// TIA Portal project "aritmetik_islemler" (V18)

(* hardware
DEVICE "S7-1200 station_1"  S7-1200 Station
   slot 0: "Rack_0"  S7-1200 Rack  Rack  V1.0
   slot 1: "PLC_1"  CPU 1214C AC/DC/Rly  6ES7 214-1BG40-0XB0  V4.6
*)

// ===== PLC "PLC_1"  CPU 1214C AC/DC/Rly =====

VAR_GLOBAL   // PLC tag table "Default tag table"
   "Tag_1" AT %I0.0 : Bool;
   "Tag_2" AT %Q0.0 : Bool;
   "Tag_3" AT %MD0 : DWord;
   "Tag_4" AT %MD8 : Real;
   "Tag_5" AT %MW2 : Int;
   "Tag_6" AT %I0.1 : Bool;
   "Tag_7" AT %M4.0 : Bool;
   "Tag_8" AT %MW8 : Int;
   "Tag_9" AT %MD16 : Real;
   "Tag_10" AT %MD12 : Real;
   "Tag_11" AT %MD24 : Real;
   "Tag_12" AT %MD20 : Real;
   "Tag_13" AT %MD10 : DWord;
END_VAR

DATA_BLOCK "Data_block_1"   // DB1
{ S7_Optimized_Access := 'TRUE' }
VERSION : 0.1
   VAR
      "A" : LReal;
      "B" : LReal;
   END_VAR
BEGIN
END_DATA_BLOCK

ORGANIZATION_BLOCK "Main"   // OB1, LAD, ProgramCycle
TITLE = "Main Program Sweep (Cycle)"
{ S7_Optimized_Access := 'TRUE' }
VERSION : 0.1
   VAR_INPUT
      Initial_Call : Bool;   // Initial call of this OB
      Remanence : Bool;   // =True, if remanent data are available
   END_VAR
   VAR_TEMP   // added for the SCL form of the ladder/FBD networks
      _w1 : Bool;
   END_VAR
BEGIN

REGION Network 1
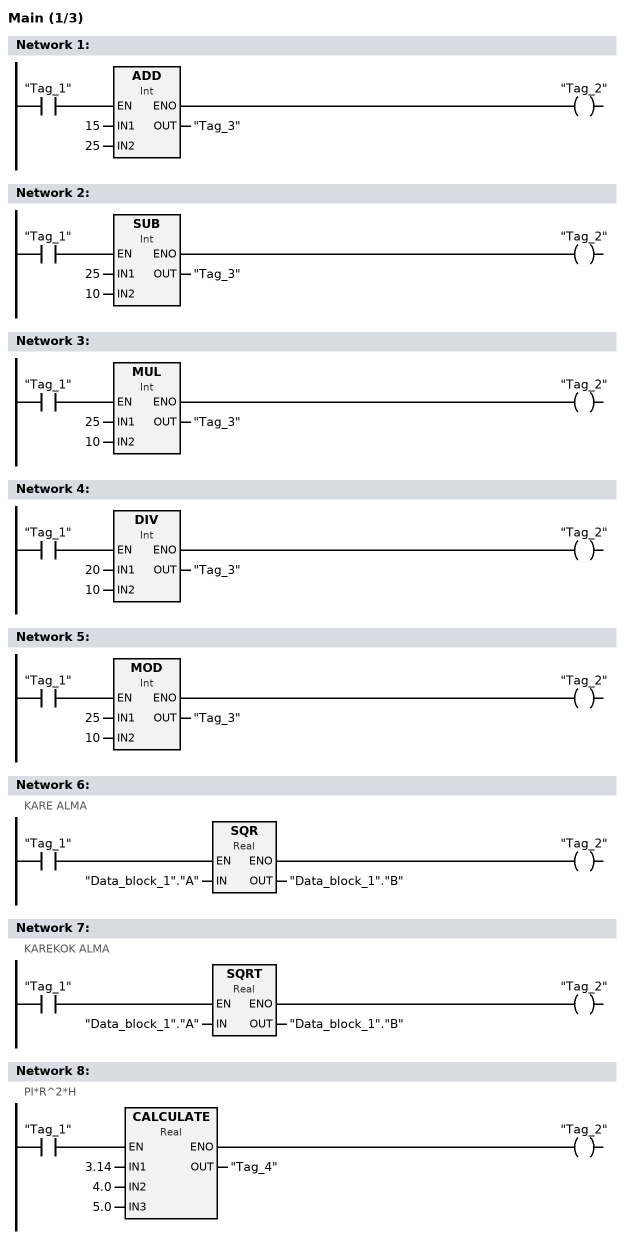
   RUNG wire#powerrail
      Contact( "Tag_1" )
      { S7_Templates := "SrcType := Int" } Add(in1 := 15, in2 := 25, out => "Tag_3")
      Coil( "Tag_2" )
   END_RUNG
   // the same network as SCL:
   IF "Tag_1" THEN "Tag_3" := 15 + 25; END_IF;
   "Tag_2" := "Tag_1";
END_REGION

REGION Network 2
   RUNG wire#powerrail
      Contact( "Tag_1" )
      { S7_Templates := "SrcType := Int" } Sub(in1 := 25, in2 := 10, out => "Tag_3")
      Coil( "Tag_2" )
   END_RUNG
   // the same network as SCL:
   IF "Tag_1" THEN "Tag_3" := 25 - 10; END_IF;
   "Tag_2" := "Tag_1";
END_REGION

REGION Network 3
   RUNG wire#powerrail
      Contact( "Tag_1" )
      { S7_Templates := "SrcType := Int" } Mul(in1 := 25, in2 := 10, out => "Tag_3")
      Coil( "Tag_2" )
   END_RUNG
   // the same network as SCL:
   IF "Tag_1" THEN "Tag_3" := 25 * 10; END_IF;
   "Tag_2" := "Tag_1";
END_REGION

REGION Network 4
   RUNG wire#powerrail
      Contact( "Tag_1" )
      { S7_Templates := "SrcType := Int" } Div(in1 := 20, in2 := 10, out => "Tag_3")
      Coil( "Tag_2" )
   END_RUNG
   // the same network as SCL:
   IF "Tag_1" THEN "Tag_3" := 20 / 10; END_IF;
   "Tag_2" := "Tag_1";
END_REGION

REGION Network 5
   RUNG wire#powerrail
      Contact( "Tag_1" )
      { S7_Templates := "SrcType := Int" } Mod(in1 := 25, in2 := 10, out => "Tag_3")
      Coil( "Tag_2" )
   END_RUNG
   // the same network as SCL:
   IF "Tag_1" THEN "Tag_3" := 25 MOD 10; END_IF;
   "Tag_2" := "Tag_1";
END_REGION

REGION Network 6
   // KARE ALMA
   IF "Tag_1" THEN "Data_block_1"."B" := SQR("Data_block_1"."A"); END_IF;
   "Tag_2" := "Tag_1";
END_REGION

REGION Network 7
   // KAREKOK ALMA
   IF "Tag_1" THEN "Data_block_1"."B" := SQRT("Data_block_1"."A"); END_IF;
   "Tag_2" := "Tag_1";
END_REGION

REGION Network 8
   // PI*R^2*H
   RUNG wire#powerrail
      Contact( "Tag_1" )
      { S7_Templates := "SrcType := Real"; S7_Expression := "IN1*(IN2*)*IN3" } Calculate(in1 := 3.14, in2 := 4.0, in3 := 5.0, out => "Tag_4")
      Coil( "Tag_2" )
   END_RUNG
   // the same network as SCL:
   // no checked SCL form for this network; see the picture
END_REGION

REGION Network 9
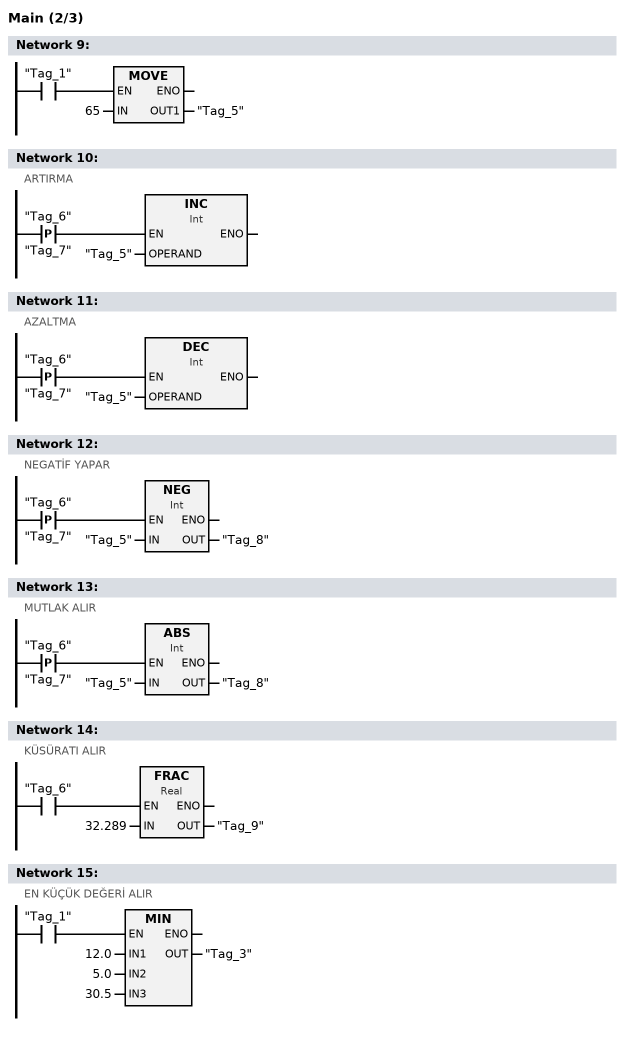
   RUNG wire#powerrail
      Contact( "Tag_1" )
      Move(in := 65, out1 => "Tag_5")
   END_RUNG
   // the same network as SCL:
   IF "Tag_1" THEN "Tag_5" := 65; END_IF;
END_REGION

REGION Network 10
   // ARTIRMA
   RUNG wire#powerrail
      P_Contact(operand := "Tag_6", bit := "Tag_7")
      { S7_Templates := "DestType := Int" } Inc( "Tag_5" )
   END_RUNG
   // the same network as SCL:
   #_w1 := "Tag_6" AND NOT "Tag_7";   // rising edge of "Tag_6"
   "Tag_7" := "Tag_6";
   IF #_w1 THEN "Tag_5" := "Tag_5" + 1; END_IF;
END_REGION

REGION Network 11
   // AZALTMA
   RUNG wire#powerrail
      P_Contact(operand := "Tag_6", bit := "Tag_7")
      { S7_Templates := "DestType := Int" } Dec( "Tag_5" )
   END_RUNG
   // the same network as SCL:
   #_w1 := "Tag_6" AND NOT "Tag_7";   // rising edge of "Tag_6"
   "Tag_7" := "Tag_6";
   IF #_w1 THEN "Tag_5" := "Tag_5" - 1; END_IF;
END_REGION

REGION Network 12
   // NEGATİF YAPAR
   RUNG wire#powerrail
      P_Contact(operand := "Tag_6", bit := "Tag_7")
      { S7_Templates := "SrcType := Int" } Neg(in := "Tag_5", out => "Tag_8")
   END_RUNG
   // the same network as SCL:
   #_w1 := "Tag_6" AND NOT "Tag_7";   // rising edge of "Tag_6"
   "Tag_7" := "Tag_6";
   IF #_w1 THEN "Tag_8" := -"Tag_5"; END_IF;
END_REGION

REGION Network 13
   // MUTLAK ALIR
   RUNG wire#powerrail
      P_Contact(operand := "Tag_6", bit := "Tag_7")
      { S7_Templates := "SrcType := Int" } Abs(in := "Tag_5", out => "Tag_8")
   END_RUNG
   // the same network as SCL:
   #_w1 := "Tag_6" AND NOT "Tag_7";   // rising edge of "Tag_6"
   "Tag_7" := "Tag_6";
   IF #_w1 THEN "Tag_8" := ABS("Tag_5"); END_IF;
END_REGION

REGION Network 14
   // KÜSÜRATI ALIR
   IF "Tag_6" THEN "Tag_9" := FRAC(32.289); END_IF;
END_REGION

REGION Network 15
   // EN KÜÇÜK DEĞERİ ALIR
   IF "Tag_1" THEN "Tag_3" := MIN(IN1 := 12.0, IN2 := 5.0, IN3 := 30.5); END_IF;
END_REGION

REGION Network 16
   // EN BÜYÜK DEĞERİ ALIR
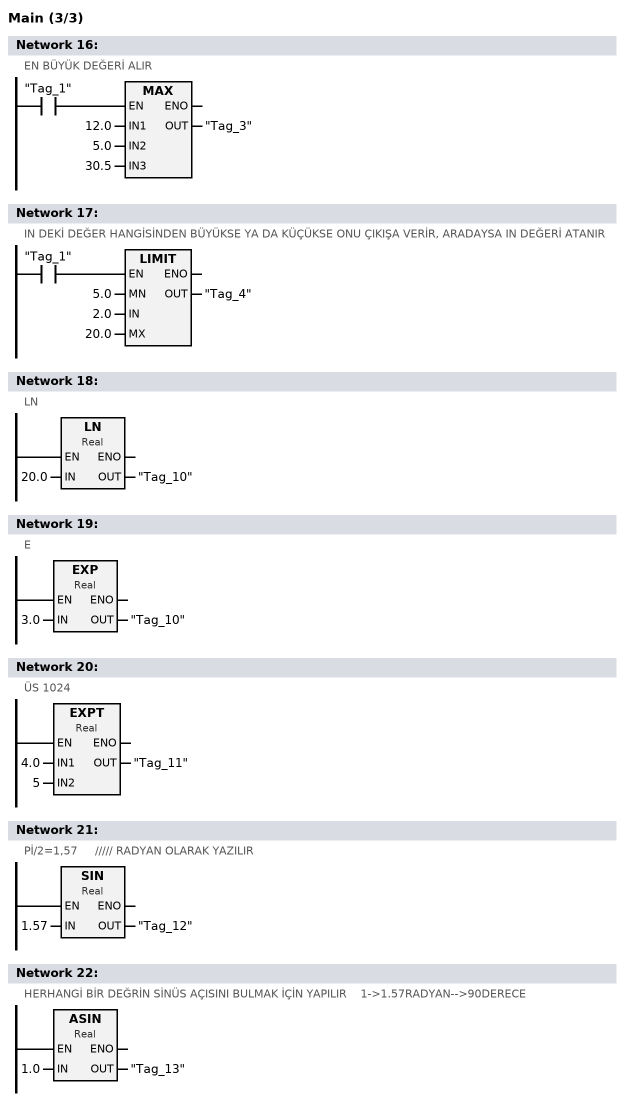
   IF "Tag_1" THEN "Tag_3" := MAX(IN1 := 12.0, IN2 := 5.0, IN3 := 30.5); END_IF;
END_REGION

REGION Network 17
   // IN DEKİ DEĞER HANGİSİNDEN BÜYÜKSE YA DA KÜÇÜKSE ONU ÇIKIŞA VERİR, ARADAYSA IN DEĞERİ ATANIR
   IF "Tag_1" THEN "Tag_4" := LIMIT(MN := 5.0, IN := 2.0, MX := 20.0); END_IF;
END_REGION

REGION Network 18
   // LN
   "Tag_10" := LN(20.0);
END_REGION

REGION Network 19
   // E
   "Tag_10" := EXP(3.0);
END_REGION

REGION Network 20
   // ÜS 1024
   "Tag_11" := 4.0 ** 5;
END_REGION

REGION Network 21
   // Pİ/2=1,57     ///// RADYAN OLARAK YAZILIR
   "Tag_12" := SIN(1.57);
END_REGION

REGION Network 22
   // HERHANGİ BİR DEĞRİN SİNÜS AÇISINI BULMAK İÇİN YAPILIR    1->1.57RADYAN-->90DERECE
   "Tag_13" := ASIN(1.0);
END_REGION
END_ORGANIZATION_BLOCK